FUNCTION_BLOCK XtsTmsTrack EXTENDS XtsTrack
VAR_INPUT
END_VAR
VAR_OUTPUT
END_VAR
VAR
	itfStartUpSequence : ITF_StartUpSequence;
END_VAR

SUPER^();

METHOD PUBLIC MoverHomeSequence : BOOL
VAR_INPUT
END_VAR
VAR
	iTmsMover : ITmsMover;
END_VAR
itfStartUpSequence.Call();
MoverHomeSequence := TRUE;
END_METHOD

PROPERTY StartSequence : ITF_StartUpSequence
GET
StartSequence := itfStartUpSequence;
END_GET
SET
itfStartUpSequence := StartSequence;
END_SET
END_PROPERTY

END_FUNCTION_BLOCK

(* stored: Version 1.1.0.1, ProductVersion 3.1.4024.11
   POU XtsTmsTrack: Id {f2eb72b4-945e-4a1d-8f0c-e37a98ea5c05}, SpecialFunc None
   Method MoverHomeSequence: Id {70291023-8adc-4c66-9169-c8ce9dca191e}
   Property StartSequence: Id {73ddcee3-e105-4b20-98c7-05fa8b502c13}
   Get Get: Id {a9047221-cfdf-4918-89b1-5f886d05b129}
   Set Set: Id {4f88209d-65f9-4fe3-be42-f9061e17a357} *)
